// TIA Portal V19 export
DATA_BLOCK "_IOL_VM_TPV70-10_Params"   // DB504
TITLE = Valve Monitoring Params for Tetra Pak V70 DeviceID: 10
{ S7_Optimized_Access := 'TRUE' }
// stored: AutoNumber false, MemoryReserve 0
   VAR RETAIN
      VM_IOL_Params : "_IOL_VM_TPV70_10";
   END_VAR
BEGIN
   VM_IOL_Params.StandardStructure.Parameter3.Subindex := 0;
END_DATA_BLOCK
